Fanuc KAREL source: kt00602.KL

-- PROVISIONAL review KL for V940-1; original PC SHA256 2c33ebf83b5687a6c96eacefc4b1ce09e903071a6308b0bace873884e0b40e82
-- Incomplete behavior may be omitted. Consult companion uncertainty JSON. Do not deploy.
PROGRAM KT00602
%NOLOCKGROUP
VAR
  I1 : INTEGER
  I2 : INTEGER
  OUT : REAL
BEGIN
  -- V9_ZERO_TABLE_METADATA_HINT layout=0001; no indexed target words; source/name/runtime held
  -- UNRESOLVED_PC offsets 5-16; opcodes 2E,23
  -- UNRESOLVED_PC offsets 21-32; opcodes 2E,23
  -- UNRESOLVED_PC offsets 37-48; opcodes 2E,23
  -- UNRESOLVED_PC offsets 53-64; opcodes 2E,23
  -- UNRESOLVED_PC offsets 69-82; opcodes 21,64,23
  -- UNRESOLVED_PC offsets 87-91; opcodes 7F
END KT00602
